TYPE struct_SFC_Row :
STRUCT
	stepName:STRING;
	AdvanceReq:BOOL;
	ReturnReq:BOOL;
	AdvanceDepth:BOOL;
	ReturnDepth:BOOL;
	
END_STRUCT
END_TYPE

(* stored: Version 1.1.0.1, ProductVersion 3.1.4024.11
   DUT struct_SFC_Row: Id {74cf5dc6-45a8-4859-932e-0c2166b8f051} *)
